% RSLogix 500 project S_ON_OFF.RSS, saved by version 7.30.10.01 %
PROJECT "S_ON_OFF"    % processor: type code 158 %

PROGRAM FILES
  LAD 2   3 rungs

DATA FILES
  O0 OUTPUT  186 elements
  I1 INPUT  130 elements
  S2 STATUS  83 elements
  B3 BINARY  1 elements
  T4 TIMER  1 elements
  C5 COUNTER  1 elements
  R6 CONTROL  1 elements
  N7 INTEGER  1 elements
  F8 FLOAT  1 elements

LADDER 2
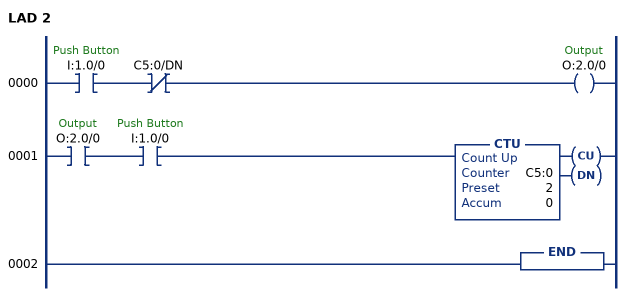
% Rung: 0 %
SOR XIC I:1.0/0 XIO C5:0/DN OTE O:2.0/0 EOR
%   I:1.0/0  "Push Button" %
%   O:2.0/0  "Output" %
% Rung: 1 %
SOR XIC O:2.0/0 XIC I:1.0/0 CTU C5:0 2 0 EOR
%   O:2.0/0  "Output" %
%   I:1.0/0  "Push Button" %
% Rung: 2 %
SOR END EOR

OTHER DOCUMENTED ADDRESSES
  O:2.0/1  "mid"
  O:2.0/2  "Output"

DATA TABLE (non-zero values as saved)
DATA C5
% .PRE .ACC %
% C5:0 % 2 0
